// TIA Portal V20 export
// export: Created 2025-12-01T14:56:27.3735686Z, ExportSetting None, DisplayName Totally Integrated Automation Portal, DisplayVersion V20 Update 3, DisplayName TIA Portal Openness, DisplayVersion V20 Update 3, DisplayName TIA Portal Version Control Interface, DisplayVersion V20 Update 3, DisplayName STEP 7 Professional, DisplayVersion V20 Update 3, DisplayName STEP 7 Safety, DisplayVersion V20 Update 2, DisplayName WinCC Basic/Comfort/Advanced, DisplayVersion V20 Update 3, DisplayName WinCC Professional, DisplayVersion V20 Update 3, DisplayName WinCC Unified, DisplayVersion V20 Update 3
ORGANIZATION_BLOCK "OB86_ERROR_SLAVES"   // OB86, LAD, RackOrStationFailure
TITLE = "Loss Of Rack Fault"
{ S7_Optimized_Access := 'FALSE' }
AUTHOR : ESTANDAR
VERSION : 3.0
// stored: SetENOAutomatically false
   VAR_TEMP
      OB86_EV_CLASS : Byte;   // 16#38/39 Event class 3
      OB86_FLT_ID : Byte;   // 16#C1/C4/C5, Fault identifcation code
      OB86_PRIORITY : Byte;   // Priority of OB Execution
      OB86_OB_NUMBR : Byte;   // 86 (Organization block 86, OB86)
      OB86_RESERVED_1 : Byte;   // Reserved for system
      OB86_RESERVED_2 : Byte;   // Reserved for system
      OB86_MDL_ADDR : Word;   // Base address of IM module in rack with fault
      OB86_Z23 : DWord;
      OB86_DATE_TIME : Date_And_Time;   // Date and time OB86 started
      P_destino : DWord;
      P_origen : DWord;
      P_infonodo : DWord;
      Numnodo : Word;
      Numred : Word;
      infonodo : Struct
         had_failed : Bool;
         deactivated : Bool;
         reserved_10 : Bool;
         reserved_11 : Bool;
         reserved_12 : Bool;
         reserved_13 : Bool;
         reserved_14 : Bool;
         reserved_15 : Bool;
         OK : Bool;
         maintenance : Bool;
         faulty : Bool;
         failed : Bool;
         was_deactivated : Bool;
         DPV1 : Bool;
         was_under_maintenance : Bool;
         was_failed : Bool;
      END_STRUCT;
   END_VAR
BEGIN
END_ORGANIZATION_BLOCK
